// TIA Portal project "Nawodnienie_tylko_zawory" (V15.1)

(* hardware
DEVICE "S7-1200 station_1"  S7-1200 Station
   slot 0: "Rack_0"  S7-1200 Rack  Rack  V1.0
   slot 1: "PLC_1"  CPU 1212C AC/DC/Rly  6ES7 212-1BE40-0XB0  V4.2
   slot 2: "DQ 8xRelay_1"  SM 1222 DQ8 x relay  6ES7 222-1HF32-0XB0  V2.0
   slot 3: "DI 2/DQ 2x24VDC_1"  DI2/DQ2 signal board (200 kHz)  6ES7 223-3BD30-0XB0  V1.0
DEVICE "HMI_1"  KP300 Basic mono PN
   slot 0: "HMI_1"  KP300 Basic mono PN  6AV6 647-0AH11-3AX0  12.0.0.0
   slot 1: "HMI_RT_1"  KP300 Basic mono PN  6AV6 647-0AH11-3AX0  12.0.0.0
   slot 5: "HMI_1.IE_CP_1"  PROFINET Interface  12.0.0.0
      slot 1: "PROFINET Interface_1"  PROFINET Interface
         slot 1: "Port_1"  Port
*)

// ===== PLC "PLC_1"  CPU 1212C AC/DC/Rly =====

VAR_GLOBAL   // PLC tag table "Output_table"
   "DQ0_III_zawor" AT %Q0.0 : Bool;
   "DQ1_II_zwor" AT %Q0.1 : Bool;
   "DQ2_I_zawor" AT %Q0.2 : Bool;
END_VAR

VAR_GLOBAL   // PLC tag table "Memory_table"
   "M0_startbutton" AT %M0.0 : Bool;
   "M01_finish_I_pole" AT %M0.1 : Bool;
   "M02_finish_II_pole" AT %M0.2 : Bool;
   "M03_finish_III_pole'" AT %M0.3 : Bool;
END_VAR

VAR_GLOBAL   // PLC tag table "Time_table"
   "T0_I_pole" AT %MD0 : Time;
   "T1_II_pole" AT %MD4 : Time;
   "T2_III_pole" AT %MD8 : Time;
END_VAR

DATA_BLOCK "Program_I_DB"   // DB1
{ S7_Optimized_Access := 'TRUE' }
VERSION : 0.1
// stored: InstanceOfName Program_I
"Program_I"
BEGIN
END_DATA_BLOCK

// folder: System blocks/Program resources

DATA_BLOCK "IEC_Timer_I_pole"   // DB5
{ S7_Optimized_Access := 'TRUE' }
AUTHOR : Simatic
FAMILY : IEC
NAME : IEC_TMR
VERSION : 1.0
// stored: InstanceOfName IEC_TIMER
"IEC_TIMER"
BEGIN
END_DATA_BLOCK

DATA_BLOCK "IEC_Timer_II_pole"   // DB6
{ S7_Optimized_Access := 'TRUE' }
AUTHOR : Simatic
FAMILY : IEC
NAME : IEC_TMR
VERSION : 1.0
// stored: InstanceOfName IEC_TIMER
"IEC_TIMER"
BEGIN
END_DATA_BLOCK

DATA_BLOCK "IEC_Timer_III_pole"   // DB7
{ S7_Optimized_Access := 'TRUE' }
AUTHOR : Simatic
FAMILY : IEC
NAME : IEC_TMR
VERSION : 1.0
// stored: InstanceOfName IEC_TIMER
"IEC_TIMER"
BEGIN
END_DATA_BLOCK

// folder: (top level)

FUNCTION_BLOCK "Program_I"   // FB1, LAD
{ S7_Optimized_Access := 'TRUE' }
VERSION : 0.1
BEGIN

REGION Network 1
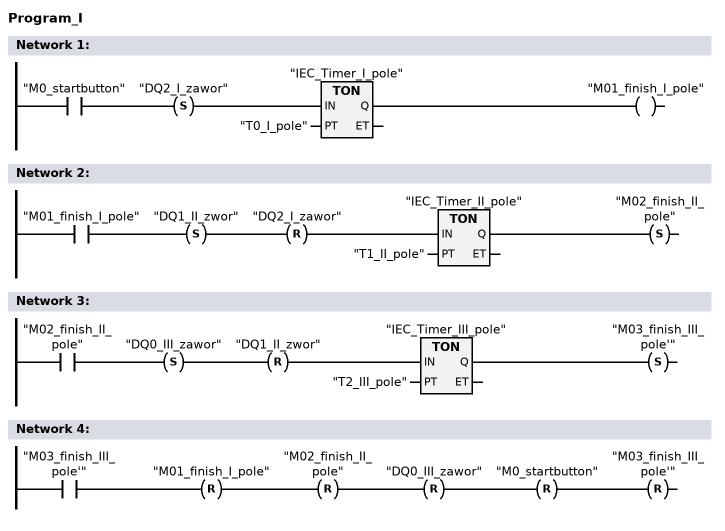
   IF "M0_startbutton" THEN "DQ2_I_zawor" := TRUE; END_IF;
   "IEC_Timer_I_pole".TON(IN := "M0_startbutton", PT := "T0_I_pole");
   "M01_finish_I_pole" := "IEC_Timer_I_pole".Q;
END_REGION

REGION Network 2
   IF "M01_finish_I_pole" THEN
       "DQ1_II_zwor" := TRUE;
       "DQ2_I_zawor" := FALSE;
   END_IF;
   "IEC_Timer_II_pole".TON(IN := "M01_finish_I_pole", PT := "T1_II_pole");
   IF "IEC_Timer_II_pole".Q THEN "M02_finish_II_pole" := TRUE; END_IF;
END_REGION

REGION Network 3
   IF "M02_finish_II_pole" THEN
       "DQ0_III_zawor" := TRUE;
       "DQ1_II_zwor" := FALSE;
   END_IF;
   "IEC_Timer_III_pole".TON(IN := "M02_finish_II_pole", PT := "T2_III_pole");
   IF "IEC_Timer_III_pole".Q THEN "M03_finish_III_pole'" := TRUE; END_IF;
END_REGION

REGION Network 4
   RUNG wire#powerrail
      Contact( "M03_finish_III_pole'" )
      R_Coil( "M01_finish_I_pole" )
      R_Coil( "M02_finish_II_pole" )
      R_Coil( "DQ0_III_zawor" )
      R_Coil( "M0_startbutton" )
      R_Coil( "M03_finish_III_pole'" )
   END_RUNG
   // the same network as SCL:
   IF "M03_finish_III_pole'" THEN
       "M01_finish_I_pole" := FALSE;
       "M02_finish_II_pole" := FALSE;
       "DQ0_III_zawor" := FALSE;
       "M0_startbutton" := FALSE;
       "M03_finish_III_pole'" := FALSE;
   END_IF;
END_REGION
END_FUNCTION_BLOCK

FUNCTION "Default_val" : Void   // FC1, SCL
{ S7_Optimized_Access := 'TRUE' }
VERSION : 0.1
BEGIN
   "T0_I_pole" := INT_TO_TIME(3) * 1000;
   "T1_II_pole" := INT_TO_TIME(3) * 1000;
   "T2_III_pole" := INT_TO_TIME(3) * 1000;
END_FUNCTION

ORGANIZATION_BLOCK "Main"   // OB1, LAD, ProgramCycle
TITLE = "Main Program Sweep (Cycle)"
{ S7_Optimized_Access := 'TRUE' }
VERSION : 0.1
   VAR_INPUT
      Initial_Call : Bool;   // Initial call of this OB
      Remanence : Bool;   // =True, if remanent data are available
   END_VAR
BEGIN

REGION Network 1
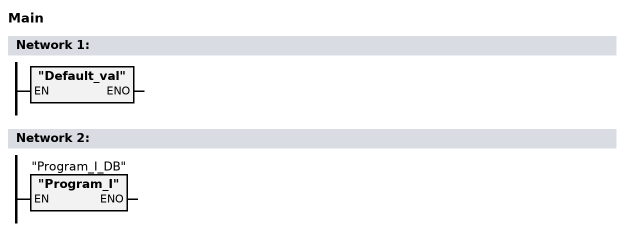
   RUNG wire#powerrail
      "Default_val"()
   END_RUNG
   // the same network as SCL:
   "Default_val"();
END_REGION

REGION Network 2
   RUNG wire#powerrail
      "Program_I_DB"()
   END_RUNG
   // the same network as SCL:
   "Program_I_DB"();   // "Program_I"
END_REGION
END_ORGANIZATION_BLOCK

(* ===== HMI "HMI_RT_1" =====

screen "Root screen" 240x80, template "Template_1"
   Button "Button_1" at 8,7 size 107x67; TextOff 'Start program'
*)